TYPE st_RegionHome :
STRUCT
	Homed	:BOOL;
	HandShake :st_HandshakeBase;
END_STRUCT
END_TYPE

(* stored: Version 1.1.0.1, ProductVersion 3.1.4024.13
   DUT st_RegionHome: Id {e538e28f-deea-4331-a292-be5f9fc512a3} *)
